(* PLC project ControlFlowFixture *)

PROGRAM CONTROL_FLOW
  VAR_INPUT
    xInitDone : BOOL;
  END_VAR

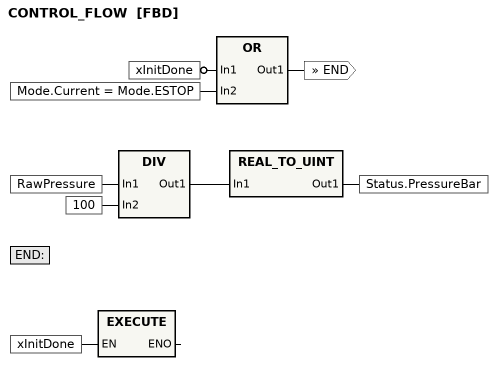
(* FBD diagram, written out as Structured Text *)
IF NOT xInitDone OR (Mode.Current = Mode.ESTOP) THEN JMP END; END_IF;
Status.PressureBar := REAL_TO_UINT(RawPressure / 100);
END:
IF xInitDone THEN
  IF NOT xInitDone THEN
  Status.PressureBar := 0;
  Status.Faulted := FALSE;
  END_IF
END_IF;
END_PROGRAM
